INTERFACE I_ControlBox

METHOD Modeselector
VAR_INPUT
END_VAR
VAR_OUTPUT
	eMode:E_Modes;
END_VAR
END_METHOD

END_INTERFACE

(* stored: Version 1.1.0.1, ProductVersion 3.1.4024.12
   Itf I_ControlBox: Id {664ffdc8-8d0d-419f-9a93-aba818157420}
   Method Modeselector: Id {139004de-a6f0-425b-b21b-ff5be7b3a2e2} *)
